TYPE TcoKukaRobotics_Status_v_5_x_x :
STRUCT
    ActionDescription : STRING(100);
    State : TcoKukaRobotics_State_v_5_x_x;
END_STRUCT
END_TYPE

(* stored: Version 1.1.0.1, ProductVersion 3.1.4024.12
   DUT TcoKukaRobotics_Status_v_5_x_x: Id {12bdb6a5-3130-0ac3-2945-23019b1e3ff4} *)
